{attribute 'TcGenerated'}
// This function has been automatically generated from the project information.
VAR_GLOBAL CONSTANT
    {attribute 'const_non_replaced'}
    {attribute 'linkalways'}
    stLibVersion_kfe_motion : ST_LibVersion := (iMajor := 1, iMinor := 4, iBuild := 1, iRevision := 0, sVersion := '1.4.1');
END_VAR

(* stored: Version 1.1.0.1, ProductVersion 3.1.4022.18
   GVL Global_Version: Id 88670457-fb1f-4346-8ddd-e8a68494c965 *)
